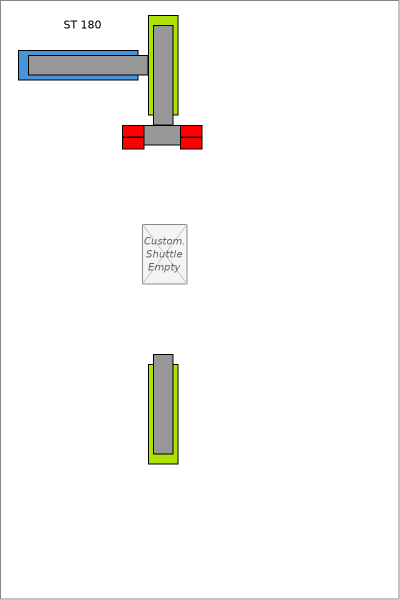
VISUALIZATION VISU_ST180  // 400x600
    Image (142,224 45x60), invisible if: NOT __ISVALIDREF(GVL.st180_aut._Mover), image: Custom.Shuttle Empty
    Rectangle (18,50 120x30)
    Rectangle (28,55 120x20)
        p3560616238: GVL.st180_aut.fb_Pnp.fb_simu_axis180_01Y.rOUT_PixActual
    Rectangle (148,15 30x100)
        p3560616238: GVL.st180_aut.fb_Pnp.fb_simu_axis180_01Y.rOUT_PixActual
    Rectangle (153,25 20x100)
        p2738717112: GVL.st180_aut.fb_Pnp.fb_simu_axis180_02Z.rOUT_PixActual
        p3560616238: GVL.st180_aut.fb_Pnp.fb_simu_axis180_01Y.rOUT_PixActual
    Label (40,15 85x20), "ST 180"
    Rectangle (122,125 80x20)
        p2738717112: GVL.st180_aut.fb_Pnp.fb_simu_axis180_02Z.rOUT_PixActual
        p3560616238: GVL.st180_aut.fb_Pnp.fb_simu_axis180_01Y.rOUT_PixActual
    Ellipse (123,125 20x20), colour toggle: GVL.st180_aut.fb_Pnp.fb_griperLeft.xIN_GS
        p3560616238: GVL.st180_aut.fb_Pnp.fb_simu_axis180_01Y.rOUT_PixActual
        p2738717112: GVL.st180_aut.fb_Pnp.fb_simu_axis180_02Z.rOUT_PixActual
    Ellipse (181,125 20x20), colour toggle: GVL.st180_aut.fb_Pnp.fb_griperRight.xIN_GS
        p3560616238: GVL.st180_aut.fb_Pnp.fb_simu_axis180_01Y.rOUT_PixActual
        p2738717112: GVL.st180_aut.fb_Pnp.fb_simu_axis180_02Z.rOUT_PixActual
    Rectangle (122,125 22x12), invisible if: NOT GVL.st180_aut.fb_Pnp.fb_clampLeft.xIN_GS
        p3560616238: GVL.st180_aut.fb_Pnp.fb_simu_axis180_01Y.rOUT_PixActual
        p2738717112: GVL.st180_aut.fb_Pnp.fb_simu_axis180_02Z.rOUT_PixActual
    Rectangle (180,125 22x12), invisible if: NOT GVL.st180_aut.fb_Pnp.fb_clampRight.xIN_GS
        p3560616238: GVL.st180_aut.fb_Pnp.fb_simu_axis180_01Y.rOUT_PixActual
        p2738717112: GVL.st180_aut.fb_Pnp.fb_simu_axis180_02Z.rOUT_PixActual
    Rectangle (122,137 22x12), invisible if: NOT GVL.st180_aut.fb_Pnp.fb_clampLeft.xIN_AS
        p3560616238: GVL.st180_aut.fb_Pnp.fb_simu_axis180_01Y.rOUT_PixActual
        p2738717112: GVL.st180_aut.fb_Pnp.fb_simu_axis180_02Z.rOUT_PixActual
    Rectangle (180,137 22x12), invisible if: NOT GVL.st180_aut.fb_Pnp.fb_clampRight.xIN_AS
        p3560616238: GVL.st180_aut.fb_Pnp.fb_simu_axis180_01Y.rOUT_PixActual
        p2738717112: GVL.st180_aut.fb_Pnp.fb_simu_axis180_02Z.rOUT_PixActual
    Rectangle (148,364 30x100)
    Rectangle (153,354 20x100)
        p2738717112: -GVL.st180_aut.fb_Pnp.fb_simu_axis180_10Z.rOUT_PixActual
END_VISUALIZATION

(* stored: Version 1.1.0.1, ProductVersion 3.1.4024.6
   Visu VISU_ST180: Id {c770e28e-aa4a-40c0-bb70-5390c2c7dda0} *)
